PROGRAM Testing
VAR
	
	StartTestSequence: BOOL;
	IterationCount	: UINT;
	RecipeID		: INT := 10001;
	
	NoOPC			: BOOL;
	state		: INT;
	OrderCnt	: UINT := 9000;
	
	TempCounter	: UINT;
END_VAR

CASE state OF
	

	0: 
		IF StartTestSequence AND NoOPC THEN
			state := 1;
		END_IF
		
	1:	
		IF Tempcounter < IterationCount THEN
			IF NOT Queue.Pending THEN
				Queue.Pending 	:= TRUE;
				Queue.RecipeID 	:= RecipeID;
				Queue.TaskID 	:= OrderCnt;
				Queue.Name		:= 'Testorder';
				Tempcounter 	:= TempCounter +1;
				OrderCnt 		:= OrderCnt +1;
				
			END_IF
		ELSE
			TempCounter 		:= 0;
			state 				:= 0;
			StartTestSequence 	:= FALSE;
		END_IF
		
		
	
	
END_CASE

END_PROGRAM

(* stored: Version 1.1.0.1, ProductVersion 3.1.0.25
   POU Testing: Id {c0a179b8-0465-4c96-87cd-56dea6ed39a3} *)
